{attribute 'GeneratedUsingTerminal: EJ1101-0022-0016'}
{attribute addProperty BoxType "EJ1101-0022-0016"}
{attribute addProperty Description "EJ1101-0022 EtherCAT Coupler (ID switch)"}
{attribute addProperty Physics "YKY"}
{attribute addProperty Id "WcStateAT %I*WcState_0B2B16F91InfoDataAT %I*InfoData_32EB74EA10"}
{attribute addProperty CRC "3571411490"}
{attribute addProperty Size "11"}
TYPE EJ1101_D4DF6A22 EXTENDS EtcSlaveBoxBase_77A0E4A7 :
STRUCT
	{attribute addProperty Name "WcState"}
	WcState : WcState_0B2B16F9;
	{attribute addProperty Name "InfoData"}
	InfoData : InfoData_32EB74EA;
END_STRUCT
END_TYPE

(* stored: Version 1.2.0.0, ProductVersion 3.1.4024.11
   DUT EJ1101_D4DF6A22: Id {84fbf41a-ad3e-4b67-a7db-55aacadfe01e} *)
